// TIA Portal project "HW_1516_reader" (V18)

(* hardware
DEVICE "S7-1500/ET200MP station_1"  S7-1500 station
   slot 0: "Rail_0"  Rack  6ES7 590-1***0-0AA0
   slot 1: "6A1"  CPU 1516-3 PN/DP  6ES7 516-3AP03-0AB0  V3.0
      slot 3: "CPU display_1"  6ES7591-1BA00-0AA0
      slot 32768: "PROFINET interface_1"  X1
         slot 32769: "Port_1"  X1 P1
         slot 32770: "Port_2"  X1 P2
      slot 33024: "PROFINET interface_2"  X2
         slot 33025: "Port_1"  X2 P1
      slot 33280: "DP interface_1"  X3
      slot 34817: "Virtual CP interface port_1"  Virtual CP interface port  Virtual CP interface port
   slot 2: "6A2"  DI 32x24VDC HF  6ES7 521-1BL00-0AB0  V2.2
   slot 3: "6A3"  AI 16xU BA  6ES7 531-7LH00-0AB0  V1.0
   slot 4: "6A4"  DO 64x24VDC/0.3A BA  6ES7 522-1BP00-0AA0  V1.0
DEVICE "GSD device_4"  GSD.Device.PN
   slot 0: "ET200SP_1"  IM 155-6 MF HF V5.2  6ES7 155-6MU00-0CN0  V5.2
      slot 0: "IM 155-6 MF HF V5.2"  IM 155-6 MF HF V5.2
      slot 1: "PN-IO"  PN-IO
   slot 0: "Rack"  Rack  V1.0
   slot 1: "DI 16x24VDC ST V1.1, QI_1"  DI 16x24VDC ST V1.1, QI  6ES7 131-6BH00-0BA0  V1.1
      slot 0: "DI 16x24VDC ST V1.1, QI"  DI 16x24VDC ST V1.1, QI
   slot 1: "Port 1 (2xFC)"  Port 1 (2xFC)  6ES7 193-6AF00-0AA0
   slot 2: "DI 16x24VDC ST V1.1, QI_2"  DI 16x24VDC ST V1.1, QI  6ES7 131-6BH00-0BA0  V1.1
      slot 0: "DI 16x24VDC ST V1.1, QI"  DI 16x24VDC ST V1.1, QI
   slot 2: "Port 2 (2xM12)"  Port 2 (2xM12)  6ES7 193-6AM00-0AA0
DEVICE "GSD device_3"  GSD.Device.PN
   slot 0: "ET200SP"  IM 155-6 PN/3 HF V4.2  6ES7 155-6AU30-0CN0  V4.2
      slot 0: "IM 155-6 PN/3 HF V4.2"  IM 155-6 PN/3 HF V4.2
      slot 1: "PN-IO"  PN-IO
   slot 0: "Rack"  Rack  V1.0
   slot 1: "DI 16x24VDC ST V1.1, QI_1"  DI 16x24VDC ST V1.1, QI  6ES7 131-6BH00-0BA0  V1.1
      slot 0: "DI 16x24VDC ST V1.1, QI"  DI 16x24VDC ST V1.1, QI
   slot 1: "Port 1 (2xRJ45)"  Port 1 (2xRJ45)  6ES7 193-6AR00-0AA0
   slot 2: "DI 16x24VDC ST V1.1, QI_2"  DI 16x24VDC ST V1.1, QI  6ES7 131-6BH00-0BA0  V1.1
      slot 0: "DI 16x24VDC ST V1.1, QI"  DI 16x24VDC ST V1.1, QI
   slot 2: "Port 2 (2xRJ45)"  Port 2 (2xRJ45)  6ES7 193-6AR00-0AA0
   slot 3: "Port 3 (2xRJ45)"  Port 3 (2xRJ45)  6ES7 193-6AR00-0AA0
   slot 4: "DI 16x24VDC ST V1.1, QI_3"  DI 16x24VDC ST V1.1, QI  6ES7 131-6BH00-0BA0  V1.1
      slot 0: "DI 16x24VDC ST V1.1, QI"  DI 16x24VDC ST V1.1, QI
DEVICE "ET 200SP station_2"  ET 200SP-Station
   slot 0: "IO device_1"  IM 155-6 PN ST  6ES7 155-6AU01-0BN0  V4.2
   slot 0: "Rack_0"  Rack  6ES5 710-8MAx1
   slot 1: "DI 8x24VDC BA_1"  DI 8x24VDC BA  6ES7 131-6BF01-0AA0  V0.0
      slot 1: "DI 8x24VDC BA_1"  DI 8x24VDC BA
   slot 2: "DI 8x24VDC BA_2"  DI 8x24VDC BA  6ES7 131-6BF01-0AA0  V0.0
      slot 1: "DI 8x24VDC BA_2"  DI 8x24VDC BA
   slot 5: "Server module_1"  Server module  6ES7 193-6PA00-0AA0  V1.1
      slot 1: "Server module_1"  Server module
   slot 127: "BA 2xRJ45"  BA 2xRJ45  6ES7 193-6AR00-0AA0  V0.0
      slot 1: "Port_1"  X1 P1 R  6ES7 193-6AR00-0AA0  V0.0
      slot 2: "Port_2"  X1 P2 R  6ES7 193-6AR00-0AA0  V0.0
DEVICE "ET 200SP station_1"  ET 200SP-Station
   slot 0: "12A1"  IM 155-6 DP HF  6ES7 155-6BU01-0CN0  V4.2
   slot 0: "Rack_0"  Rack  6ES5 710-8MAx1
   slot 1: "12A2"  DI 8x24VDC BA  6ES7 131-6BF01-0AA0  V0.0
      slot 1: "12A2"  DI 8x24VDC BA
   slot 2: "12A3"  DI 8x24VDC BA  6ES7 131-6BF01-0AA0  V0.0
      slot 1: "12A3"  DI 8x24VDC BA
   slot 3: "12A4"  DQ 16x24VDC/0.5A BA  6ES7 132-6BH00-0AA0  V0.0
      slot 1: "12A4"  DQ 16x24VDC/0.5A BA
   slot 4: "Server module_1"  Server module  6ES7 193-6PA00-0AA0  V1.1
      slot 1: "Server module_1"  Server module
DEVICE "GSD device_1"  GSD.Device.PN
   slot 0: "11A1"  IM 155-6 PN ST V3.3  6ES7 155-6AU00-0BN0  V3.3
      slot 0: "IM 155-6 PN ST V3.3"  IM 155-6 PN ST V3.3
      slot 1: "PN-IO"  PN-IO
   slot 0: "Rack"  Rack  V1.0
   slot 1: "11A2"  DI 8x24VDC ST V1.1  6ES7 131-6BF00-0BA0  V1.1
      slot 0: "DI 8x24VDC ST V1.1"  DI 8x24VDC ST V1.1
   slot 1: "Port 1 (2xRJ45)"  Port 1 (2xRJ45)  6ES7 193-6AR00-0AA0
   slot 2: "11A3"  DI 8x24VDC ST V1.1  6ES7 131-6BF00-0BA0  V1.1
      slot 0: "DI 8x24VDC ST V1.1"  DI 8x24VDC ST V1.1
   slot 2: "Port 2 (2xRJ45)"  Port 2 (2xRJ45)  6ES7 193-6AR00-0AA0
   slot 3: "11A4"  DQ 8x24VDC/0.5A ST V1.1  6ES7 132-6BF00-0BA0  V1.1
      slot 0: "DQ 8x24VDC/0.5A ST V1.1"  DQ 8x24VDC/0.5A ST V1.1
DEVICE "GSD device_2"  GSD.Device.PN
   slot 0: "10A1"  DataMan 280 CC-B  DMR-28x-xx  6.2.0
      slot 0: "DataMan 280 CC-B"  DataMan 280 CC-B
      slot 1: "Interface"  Interface
         slot 1: "Port 1"  Port 1
   slot 0: "Rack"  Rack  V1.0
   slot 1: "Acquisition Control_1"  Acquisition Control
      slot 0: "Acquisition Control"  Acquisition Control
   slot 2: "Acquisition Status_1"  Acquisition Status
      slot 0: "Acquisition Status"  Acquisition Status
   slot 3: "Results Control_1"  Results Control
      slot 0: "Results Control"  Results Control
   slot 4: "Results Status_1"  Results Status
      slot 0: "Results Status"  Results Status
   slot 5: "Soft Event Control_1"  Soft Event Control
      slot 0: "Soft Event Control"  Soft Event Control
   slot 6: "User Data - 64 bytes_1"  User Data - 64 bytes
      slot 0: "User Data - 64 bytes"  User Data - 64 bytes
   slot 7: "Result Data - 64 bytes_1"  Result Data - 64 bytes
      slot 0: "Result Data - 64 bytes"  Result Data - 64 bytes
*)

// ===== PLC "6A1"  CPU 1516-3 PN/DP =====

VAR_GLOBAL   // PLC tag table "Default tag table"
   "Clock_Byte" AT %MB0 : Byte;
   "Clock_10Hz" AT %M0.0 : Bool;
   "Clock_5Hz" AT %M0.1 : Bool;
   "Clock_2.5Hz" AT %M0.2 : Bool;
   "Clock_2Hz" AT %M0.3 : Bool;
   "Clock_1.25Hz" AT %M0.4 : Bool;
   "Clock_1Hz" AT %M0.5 : Bool;
   "Clock_0.625Hz" AT %M0.6 : Bool;
   "Clock_0.5Hz" AT %M0.7 : Bool;
   "System_Byte" AT %MB1 : Byte;
   "FirstScan" AT %M1.0 : Bool;
   "DiagStatusUpdate" AT %M1.1 : Bool;
   "AlwaysTRUE" AT %M1.2 : Bool;
   "AlwaysFALSE" AT %M1.3 : Bool;
END_VAR

ORGANIZATION_BLOCK "Main"   // OB1, LAD, ProgramCycle
TITLE = "Main Program Sweep (Cycle)"
{ S7_Optimized_Access := 'TRUE' }
VERSION : 0.1
   VAR_INPUT
      Initial_Call : Bool;   // Initial call of this OB
      Remanence : Bool;   // =True, if remanent data are available
   END_VAR
BEGIN
END_ORGANIZATION_BLOCK